FUNCTION FB_Check : BOOL
VAR_INPUT
END_VAR
VAR
END_VAR

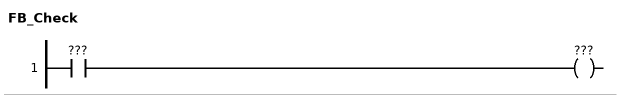
// NETWORK 1
??? := ???;

END_FUNCTION

(* stored: Version 1.1.0.1, ProductVersion 3.1.4024.11
   POU FB_Check: Id {74730271-9b70-0483-1437-09d76558bc14}, SpecialFunc None *)
